ABB RAPID module: MainModule.mod

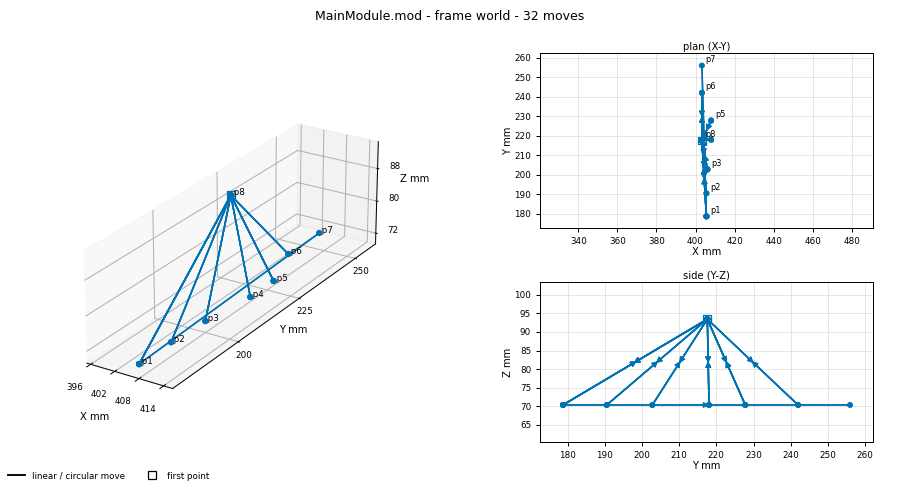
[picture p0: tool path of MainModule.mod in frame world, 32 of 32 moves have a stored position in this frame; points joined in program order, loops and branches not executed]
MODULE MainModule
    LOCAL CONST string YuMi_App_Program_Version:="1.0.1"; !Do not edit or remove this line!
	LOCAL CONST robtarget p49:=[[392.87,10.18,52.15],[0.174306,-0.285862,0.880906,-0.334522],[-1,2,-1,4],[120.635,9E+09,9E+09,9E+09,9E+09,9E+09]];
	LOCAL VAR robtarget p0:=[[195.05,297.75,84.84],[0.272693,0.635761,0.62248,0.366012],[0,0,-1,4],[98.0726,9E+09,9E+09,9E+09,9E+09,9E+09]];
	LOCAL VAR robtarget p10:=[[195.02,297.75,84.82],[0.271625,0.635189,0.622956,0.366988],[0,0,-1,4],[98.0728,9E+09,9E+09,9E+09,9E+09,9E+09]];
	LOCAL CONST robtarget p59:=[[195.02,297.75,84.82],[0.271624,0.635191,0.622955,0.366987],[0,0,-1,4],[98.0728,9E+09,9E+09,9E+09,9E+09,9E+09]];
    LOCAL VAR robtarget p48:=[[436.52,5.22,67.79],[0.301532,-0.282635,0.784603,-0.462162],[-1,2,-1,4],[120.792,9E+09,9E+09,9E+09,9E+09,9E+09]];
    LOCAL VAR robtarget p47:=[[434.08,5.22,267.93],[0.301536,-0.282667,0.784604,-0.462138],[-1,2,-1,4],[120.792,9E+09,9E+09,9E+09,9E+09,9E+09]];
    LOCAL VAR robtarget p1:=[[405.58,178.76,70.37],[0.302709,-0.2827,0.783782,-0.462746],[-1,0,1,4],[145.628,9E+09,9E+09,9E+09,9E+09,9E+09]];
    LOCAL VAR robtarget p2:=[[405.58,190.54,70.37],[0.302683,-0.282688,0.783798,-0.462744],[-1,0,1,4],[145.627,9E+09,9E+09,9E+09,9E+09,9E+09]];
    LOCAL VAR robtarget p3:=[[406.17,202.80,70.37],[0.302726,-0.282692,0.783783,-0.462738],[-1,0,1,4],[145.627,9E+09,9E+09,9E+09,9E+09,9E+09]];
    LOCAL VAR robtarget p4:=[[407.97,218.04,70.37],[0.302758,-0.282696,0.783779,-0.462721],[-1,0,1,4],[145.627,9E+09,9E+09,9E+09,9E+09,9E+09]];
    LOCAL VAR robtarget p5:=[[407.98,227.79,70.37],[0.302766,-0.282695,0.783778,-0.462718],[-1,0,1,4],[145.627,9E+09,9E+09,9E+09,9E+09,9E+09]];
    LOCAL VAR robtarget p6:=[[403.27,241.99,70.37],[0.302767,-0.282695,0.783778,-0.462718],[-1,0,1,4],[145.627,9E+09,9E+09,9E+09,9E+09,9E+09]];
    LOCAL VAR robtarget p7:=[[403.27,255.96,70.37],[0.302761,-0.28269,0.783784,-0.462715],[-1,0,1,4],[145.626,9E+09,9E+09,9E+09,9E+09,9E+09]];
    LOCAL VAR robtarget p8:=[[403.29,217.58,93.45],[0.302805,-0.282682,0.783773,-0.462709],[-1,0,1,4],[145.627,9E+09,9E+09,9E+09,9E+09,9E+09]];
	PROC main()
        MoveL p8, v200, z0, YuMi_App_move_tool_local;
        MoveL p1, v50, z0, YuMi_App_move_tool_local;
        MoveL p7, v50, z0, YuMi_App_move_tool_local;
        MoveL p1, v50, z0, YuMi_App_move_tool_local;
        MoveL p8, v200, z0, YuMi_App_move_tool_local;
		MoveL p1, v200, z0, YuMi_App_move_tool_local;
        MoveL p8, v200, z0, YuMi_App_move_tool_local;
		MoveL p1, v200, z0, YuMi_App_move_tool_local;
        MoveL p8, v200, z0, YuMi_App_move_tool_local;
        MoveL p5, v200, z0, YuMi_App_move_tool_local;
        MoveL p8, v200, z0, YuMi_App_move_tool_local;
		MoveL p5, v200, z0, YuMi_App_move_tool_local;
        MoveL p8, v200, z0, YuMi_App_move_tool_local;
        MoveL p6, v200, z0, YuMi_App_move_tool_local;
        MoveL p8, v200, z0, YuMi_App_move_tool_local;
		MoveL p6, v200, z0, YuMi_App_move_tool_local;
        MoveL p8, v200, z0, YuMi_App_move_tool_local;
        MoveL p5, v200, z0, YuMi_App_move_tool_local;
        MoveL p8, v200, z0, YuMi_App_move_tool_local;
		MoveL p4, v200, z0, YuMi_App_move_tool_local;
        MoveL p8, v200, z0, YuMi_App_move_tool_local;
        MoveL p4, v200, z0, YuMi_App_move_tool_local;
        MoveL p8, v200, z0, YuMi_App_move_tool_local;
		MoveL p3, v200, z0, YuMi_App_move_tool_local;
        MoveL p8, v200, z0, YuMi_App_move_tool_local;
        MoveL p3, v200, z0, YuMi_App_move_tool_local;
        MoveL p8, v200, z0, YuMi_App_move_tool_local;
		MoveL p2, v200, z0, YuMi_App_move_tool_local;
        MoveL p8, v200, z0, YuMi_App_move_tool_local;
        MoveL p2, v200, z0, YuMi_App_move_tool_local;
        MoveL p8, v200, z0, YuMi_App_move_tool_local;
		MoveL p1, v200, z0, YuMi_App_move_tool_local;
       ! MoveL p0, v200, z50, YuMi_App_move_tool_local;
	!MoveL p48, v200, z50, YuMi_App_move_tool_local;
	 !  SetDO Gripper,1;  ! Set the output to open the gripper
     !  WaitTime 0.5;           ! Wait for the gripper to fully open
     !  SetDO gripper_close, 0; ! Ensure close command is off
	ENDPROC
ENDMODULE
